(* Logix 5000 project; controller STAT 1756-L72 rev 20.12; software revision 20.04; part 34 of 34 *)
(* tags used below, declared in another part *)
   B3 : DINT[50];
   F8 : REAL[200];
   I1_000_Bit09 : ALIAS FOR stock:1:I.Point_9;
   I1_000_Bit10 : ALIAS FOR stock:1:I.Point_10;
   I2_000_Bit13 : ALIAS FOR stock:2:I.Point_13;   // chaudière colmatageLigne 30= on 1= off
   I2_000_Bit14 : ALIAS FOR stock:2:I.Point_14;   // DEFAUT CHAUDIEREiwts
   N20 : DINT[100];
   N7 : DINT[255];
   nitric_occupe : BOOL;
   O3_000_Bit06 : ALIAS FOR stock:3:O.Point_6;   // lampe BP sur ligne p
   O3_000_Bit07 : ALIAS FOR stock:3:O.Point_7;
   ons11 : BOOL;
   S_bp_dmd_naoh : BOOL;
   S_ok_pmp_nitrique : BOOL;
   S_run_pmp_nitrique : BOOL;
   T4 : TIMER[50];
   apport_soude_ibt_occupe : BOOL;
   dmd_soude_ibt_ok : BOOL;
   I19_001_Bit07 : ALIAS FOR I19[1].7;   // vanne soude de stock ouverte
   I19_001_Bit08 : ALIAS FOR I19[1].8;   // vanne soude de stock fermée
   L1_stat : DINT[20];
   L2_STAT : DINT[20];
   L3_STAT : DINT[20];
   lancystock1 : DINT;
   lancystock2 : DINT;
   MSG_R_L4 : MESSAGE;
   MSG_W_L4 : MESSAGE;
   mw2 : BOOL;
   N : INT[255];
   O16 : INT[2];
   onS14 : BOOL;
   onS15 : BOOL;
   onS16 : BOOL;
   S_def_airco_hT_l1 : BOOL;
   S_def_ventilo_hT_l1 : BOOL;
   S_naoh_ibt : BOOL;
   S_stock_v_naoh_f : BOOL;
   S_stock_v_naoh_o : BOOL;
   soude_ibt_fini : BOOL;
   stat_L1 : DINT[20];
   STAT_L2 : DINT[20];
   STAT_L3 : DINT[20];
   stocklancy1 : DINT;
   stocklancy2 : DINT;
   stocklancy4 : DINT;   // alarme lvl 1 stock
   stocklancy5 : DINT;   // alarme lvl 2 stock
   t1sec : TIMER;
(* stock, continued *)

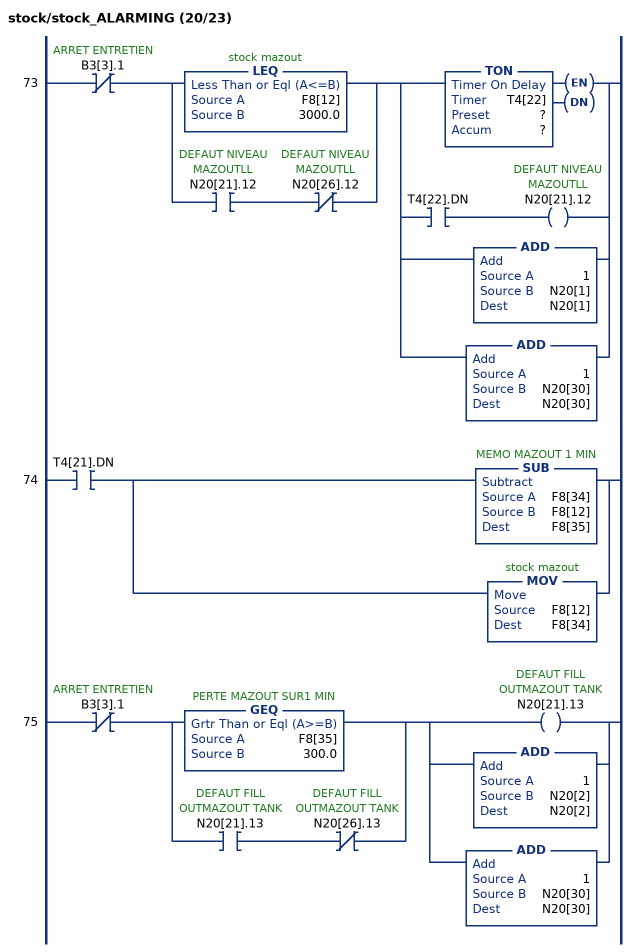
   [picture p698: stock/stock_ALARMING rungs 73-75]
   73: XIO(B3[3].1)[LEQ(F8[12],3000.0) ,XIC(N20[21].12) XIO(N20[26].12) ][TON(T4[22],?,?) ,XIC(T4[22].DN) OTE(N20[21].12) ,ADD(1,N20[1],N20[1]) ,ADD(1,N20[30],N20[30]) ];
   74: XIC(T4[21].DN)[SUB(F8[34],F8[12],F8[35]) ,MOV(F8[12],F8[34]) ];
   75: XIO(B3[3].1)[GEQ(F8[35],300.0) ,XIC(N20[21].13) XIO(N20[26].13) ][OTE(N20[21].13) ,ADD(1,N20[2],N20[2]) ,ADD(1,N20[30],N20[30]) ];
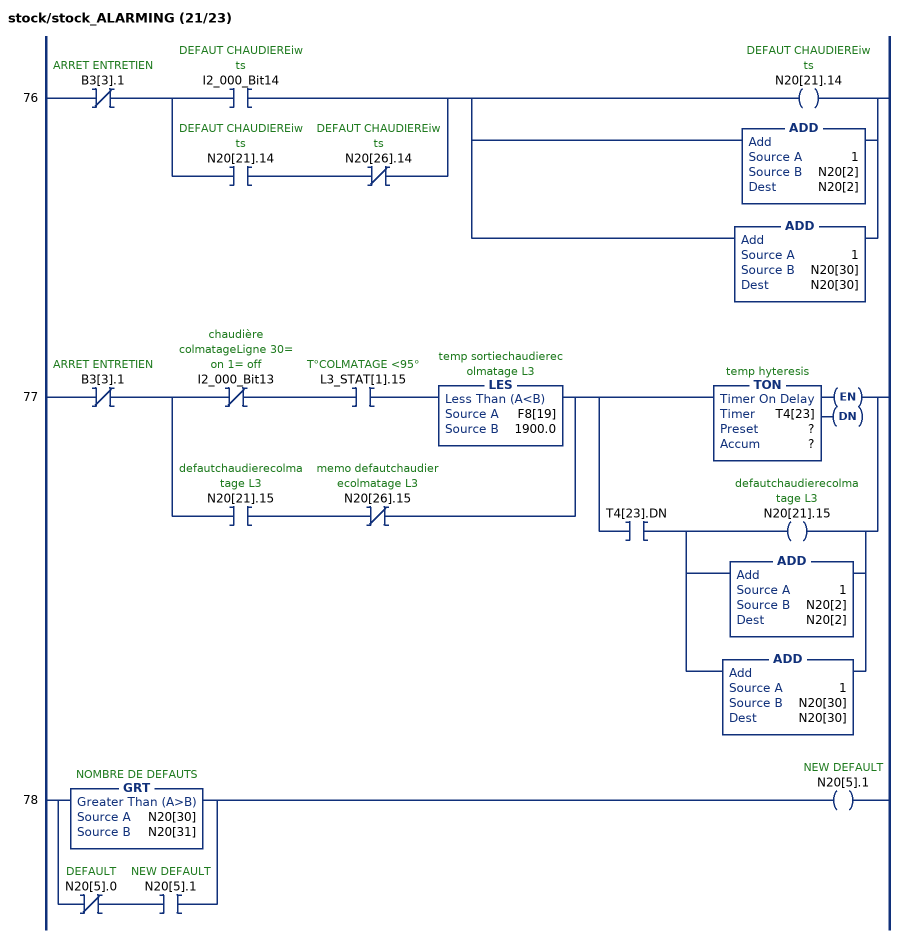
   76: XIO(B3[3].1)[XIC(I2_000_Bit14) ,XIC(N20[21].14) XIO(N20[26].14) ][OTE(N20[21].14) ,ADD(1,N20[2],N20[2]) ,ADD(1,N20[30],N20[30]) ];
   77: XIO(B3[3].1)[XIO(I2_000_Bit13) XIC(L3_STAT[1].15) LES(F8[19],1900.0) ,XIC(N20[21].15) XIO(N20[26].15) ][TON(T4[23],?,?) ,XIC(T4[23].DN) [OTE(N20[21].15) ,ADD(1,N20[2],N20[2]) ,ADD(1,N20[30],N20[30]) ] ];
   78: [GRT(N20[30],N20[31]) ,XIO(N20[5].0) XIC(N20[5].1) ]OTE(N20[5].1);
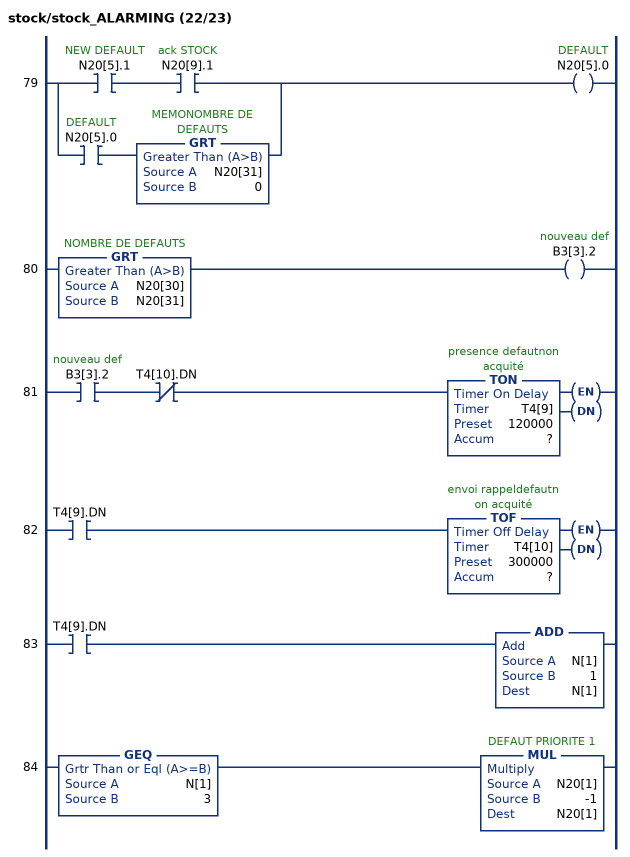
   79: [XIC(N20[5].1) XIC(N20[9].1) ,XIC(N20[5].0) GRT(N20[31],0) ]OTE(N20[5].0);
   80: GRT(N20[30],N20[31])OTE(B3[3].2);
   81: XIC(B3[3].2)XIO(T4[10].DN)TON(T4[9],?,?);
   82: XIC(T4[9].DN)TOF(T4[10],?,?);
   83: XIC(T4[9].DN)ADD(N[1],1,N[1]);
   84: GEQ(N[1],3)MUL(N20[1],-1,N20[1]);
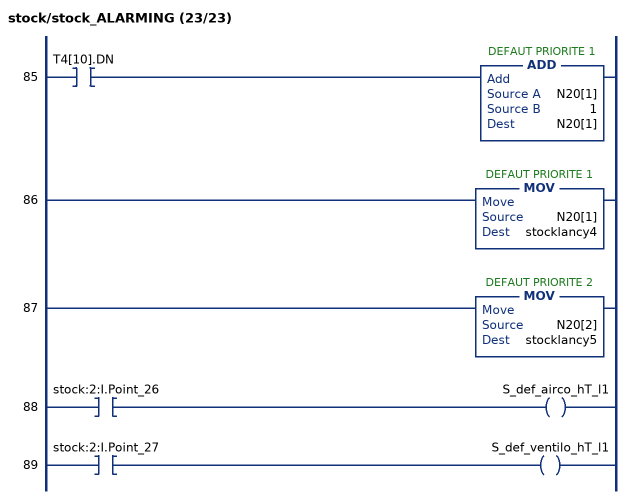
   85: XIC(T4[10].DN)ADD(N20[1],1,N20[1]);
   86: MOV(N20[1],stocklancy4);
   87: MOV(N20[2],stocklancy5);
   88: XIC(stock:2:I.Point_26)OTE(S_def_airco_hT_l1);
   89: XIC(stock:2:I.Point_27)OTE(S_def_ventilo_hT_l1);
END_ROUTINE

ROUTINE stock_nitric   (* ladder *)
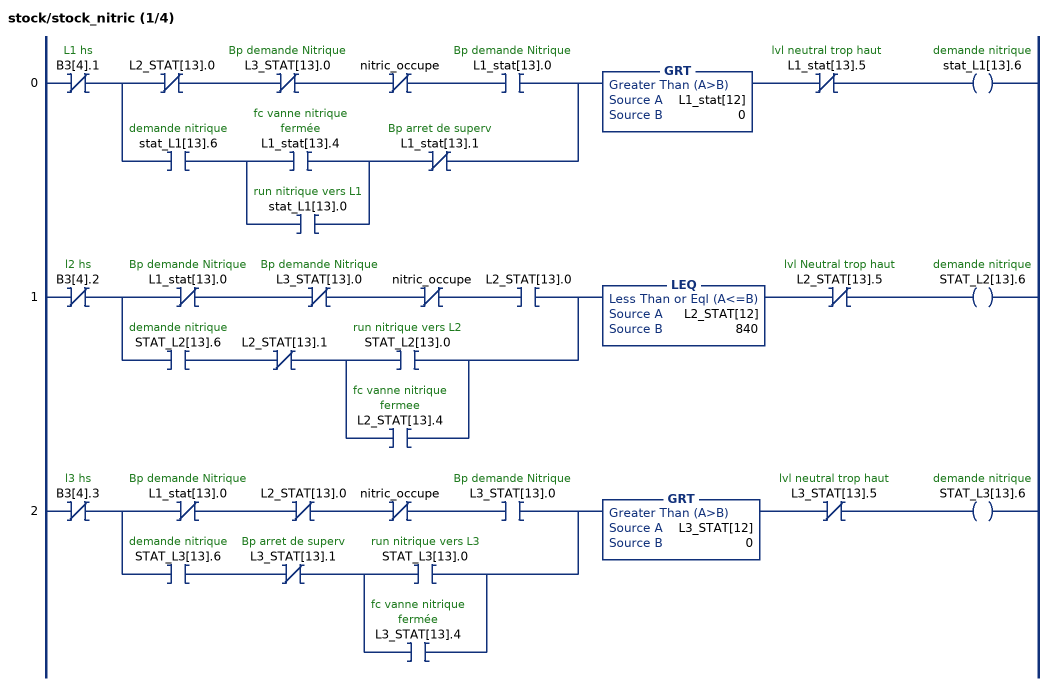
   0: XIO(B3[4].1)[XIO(L2_STAT[13].0) XIO(L3_STAT[13].0) XIO(nitric_occupe) XIC(L1_stat[13].0) ,XIC(stat_L1[13].6) [XIC(L1_stat[13].4) ,XIC(stat_L1[13].0) ] XIO(L1_stat[13].1) ]GRT(L1_stat[12],0)XIO(L1_stat[13].5)OTE(stat_L1[13].6);
   1: XIO(B3[4].2)[XIO(L1_stat[13].0) XIO(L3_STAT[13].0) XIO(nitric_occupe) XIC(L2_STAT[13].0) ,XIC(STAT_L2[13].6) XIO(L2_STAT[13].1) [XIC(STAT_L2[13].0) ,XIC(L2_STAT[13].4) ] ]LEQ(L2_STAT[12],840)XIO(L2_STAT[13].5)OTE(STAT_L2[13].6);
   2: XIO(B3[4].3)[XIO(L1_stat[13].0) XIO(L2_STAT[13].0) XIO(nitric_occupe) XIC(L3_STAT[13].0) ,XIC(STAT_L3[13].6) XIO(L3_STAT[13].1) [XIC(STAT_L3[13].0) ,XIC(L3_STAT[13].4) ] ]GRT(L3_STAT[12],0)XIO(L3_STAT[13].5)OTE(STAT_L3[13].6);
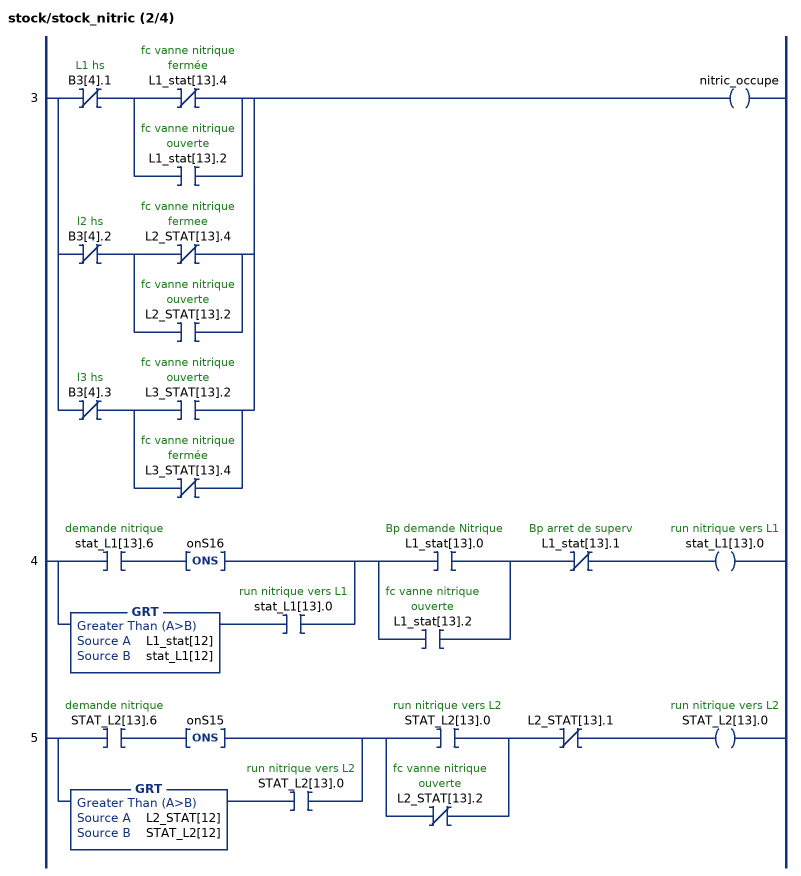
   3: [XIO(B3[4].1) [XIO(L1_stat[13].4) ,XIC(L1_stat[13].2) ] ,XIO(B3[4].2) [XIO(L2_STAT[13].4) ,XIC(L2_STAT[13].2) ] ,XIO(B3[4].3) [XIC(L3_STAT[13].2) ,XIO(L3_STAT[13].4) ] ]OTE(nitric_occupe);
   4: [XIC(stat_L1[13].6) ONS(onS16) ,GRT(L1_stat[12],stat_L1[12]) XIC(stat_L1[13].0) ][XIC(L1_stat[13].0) ,XIC(L1_stat[13].2) ]XIO(L1_stat[13].1)OTE(stat_L1[13].0);
   5: [XIC(STAT_L2[13].6) ONS(onS15) ,GRT(L2_STAT[12],STAT_L2[12]) XIC(STAT_L2[13].0) ][XIC(STAT_L2[13].0) ,XIO(L2_STAT[13].2) ]XIO(L2_STAT[13].1)OTE(STAT_L2[13].0);
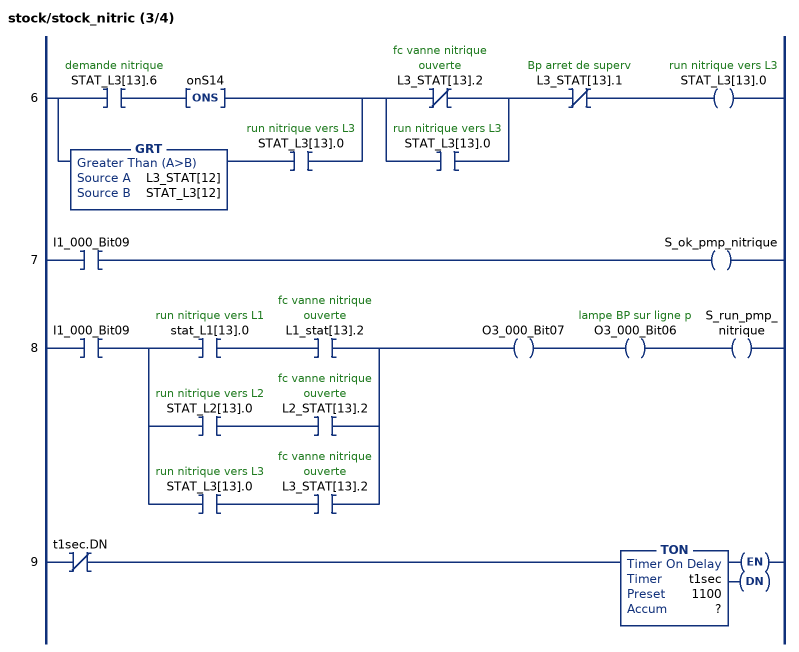
   6: [XIC(STAT_L3[13].6) ONS(onS14) ,GRT(L3_STAT[12],STAT_L3[12]) XIC(STAT_L3[13].0) ][XIO(L3_STAT[13].2) ,XIC(STAT_L3[13].0) ]XIO(L3_STAT[13].1)OTE(STAT_L3[13].0);
   7: XIC(I1_000_Bit09)OTE(S_ok_pmp_nitrique);
   8: XIC(I1_000_Bit09)[XIC(stat_L1[13].0) XIC(L1_stat[13].2) ,XIC(STAT_L2[13].0) XIC(L2_STAT[13].2) ,XIC(STAT_L3[13].0) XIC(L3_STAT[13].2) ]OTE(O3_000_Bit07)OTE(O3_000_Bit06)OTE(S_run_pmp_nitrique);
   9: XIO(t1sec.DN)TON(t1sec,?,?);
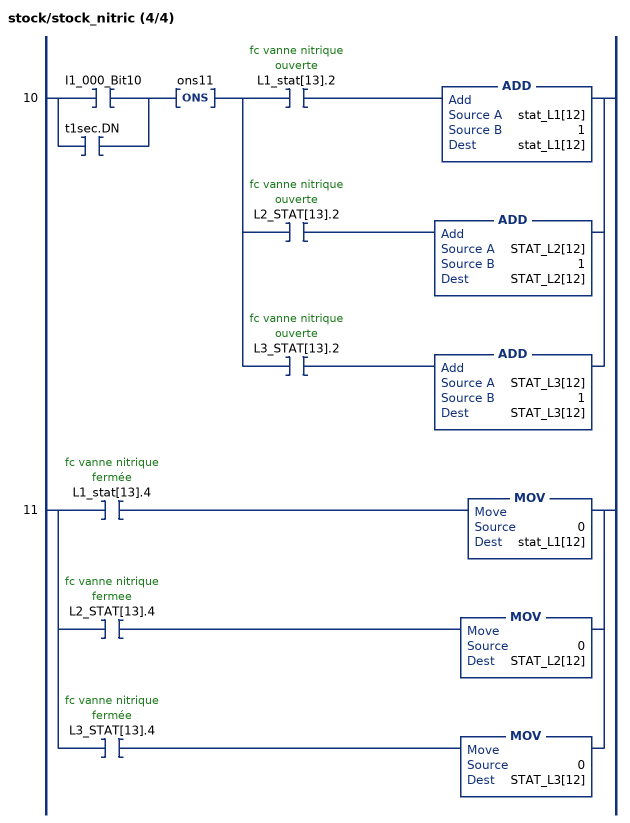
   10: [XIC(I1_000_Bit10) ,XIC(t1sec.DN) ]ONS(ons11)[XIC(L1_stat[13].2) ADD(stat_L1[12],1,stat_L1[12]) ,XIC(L2_STAT[13].2) ADD(STAT_L2[12],1,STAT_L2[12]) ,XIC(L3_STAT[13].2) ADD(STAT_L3[12],1,STAT_L3[12]) ];
   11: [XIC(L1_stat[13].4) MOV(0,stat_L1[12]) ,XIC(L2_STAT[13].4) MOV(0,STAT_L2[12]) ,XIC(L3_STAT[13].4) MOV(0,STAT_L3[12]) ];
END_ROUTINE

ROUTINE stock_SOUDE   (* ladder *)
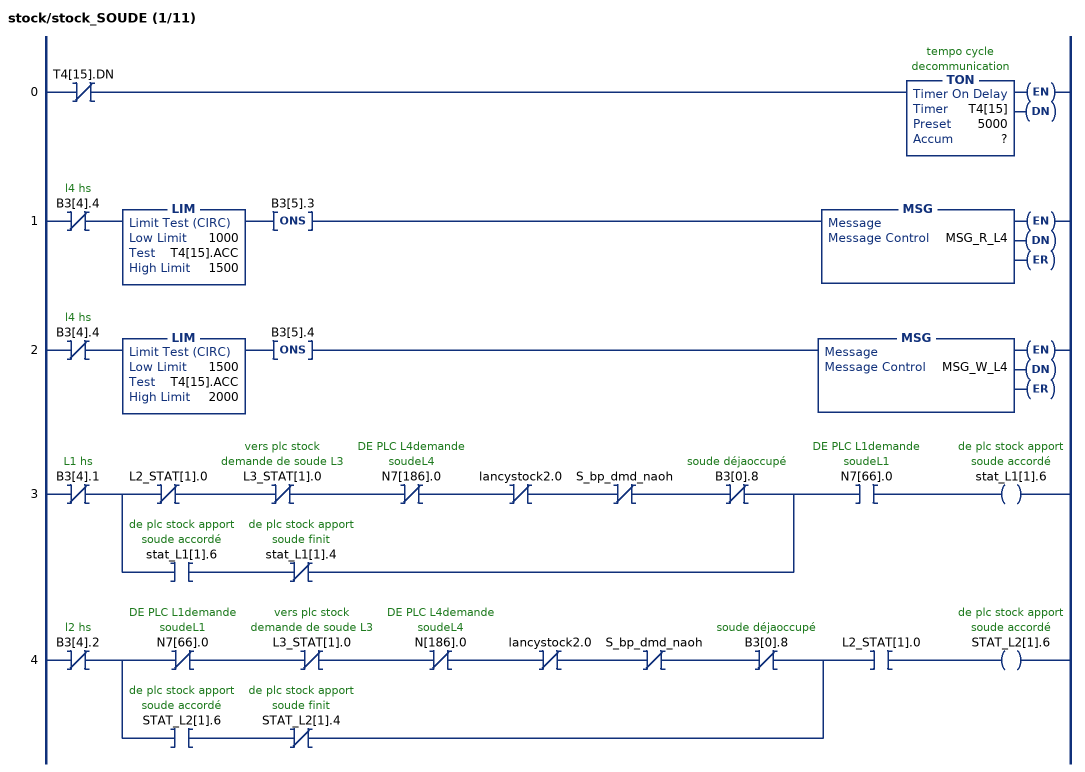
   0: XIO(T4[15].DN)TON(T4[15],?,?);
   1: XIO(B3[4].4)LIM(1000,T4[15].ACC,1500)ONS(B3[5].3)MSG(MSG_R_L4);
   2: XIO(B3[4].4)LIM(1500,T4[15].ACC,2000)ONS(B3[5].4)MSG(MSG_W_L4);
   3: XIO(B3[4].1)[XIO(L2_STAT[1].0) XIO(L3_STAT[1].0) XIO(N7[186].0) XIO(lancystock2.0) XIO(S_bp_dmd_naoh) XIO(B3[0].8) ,XIC(stat_L1[1].6) XIO(stat_L1[1].4) ]XIC(N7[66].0)OTE(stat_L1[1].6);
   4: XIO(B3[4].2)[XIO(N7[66].0) XIO(L3_STAT[1].0) XIO(N[186].0) XIO(lancystock2.0) XIO(S_bp_dmd_naoh) XIO(B3[0].8) ,XIC(STAT_L2[1].6) XIO(STAT_L2[1].4) ]XIC(L2_STAT[1].0)OTE(STAT_L2[1].6);
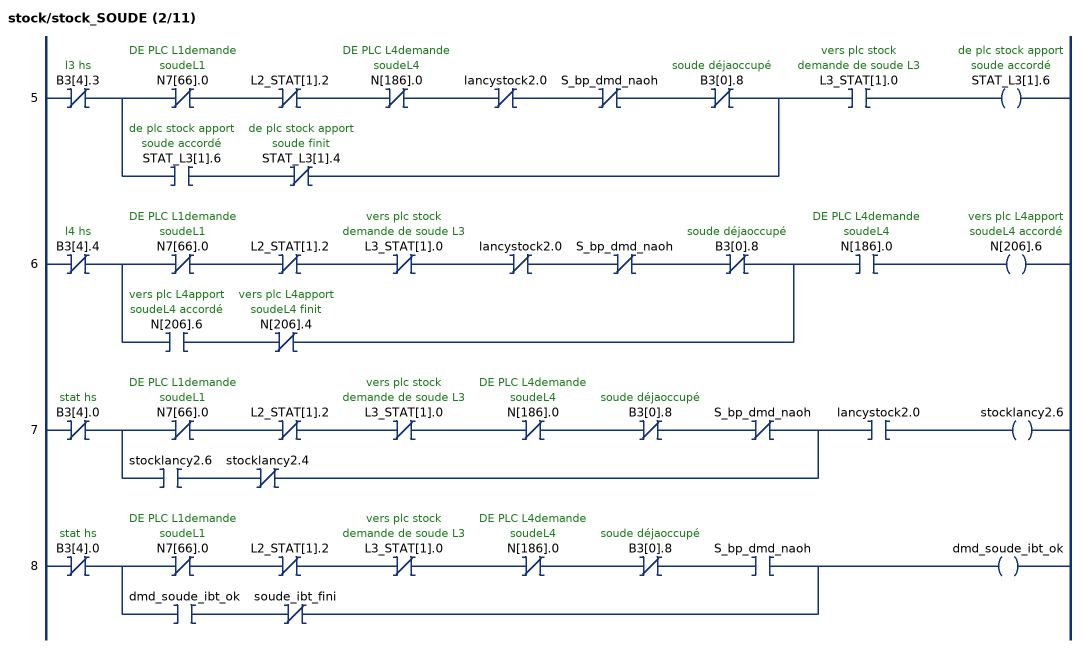
   5: XIO(B3[4].3)[XIO(N7[66].0) XIO(L2_STAT[1].2) XIO(N[186].0) XIO(lancystock2.0) XIO(S_bp_dmd_naoh) XIO(B3[0].8) ,XIC(STAT_L3[1].6) XIO(STAT_L3[1].4) ]XIC(L3_STAT[1].0)OTE(STAT_L3[1].6);
   6: XIO(B3[4].4)[XIO(N7[66].0) XIO(L2_STAT[1].2) XIO(L3_STAT[1].0) XIO(lancystock2.0) XIO(S_bp_dmd_naoh) XIO(B3[0].8) ,XIC(N[206].6) XIO(N[206].4) ]XIC(N[186].0)OTE(N[206].6);
   7: XIO(B3[4].0)[XIO(N7[66].0) XIO(L2_STAT[1].2) XIO(L3_STAT[1].0) XIO(N[186].0) XIO(B3[0].8) XIO(S_bp_dmd_naoh) ,XIC(stocklancy2.6) XIO(stocklancy2.4) ]XIC(lancystock2.0)OTE(stocklancy2.6);
   8: XIO(B3[4].0)[XIO(N7[66].0) XIO(L2_STAT[1].2) XIO(L3_STAT[1].0) XIO(N[186].0) XIO(B3[0].8) XIC(S_bp_dmd_naoh) ,XIC(dmd_soude_ibt_ok) XIO(soude_ibt_fini) ]OTE(dmd_soude_ibt_ok);
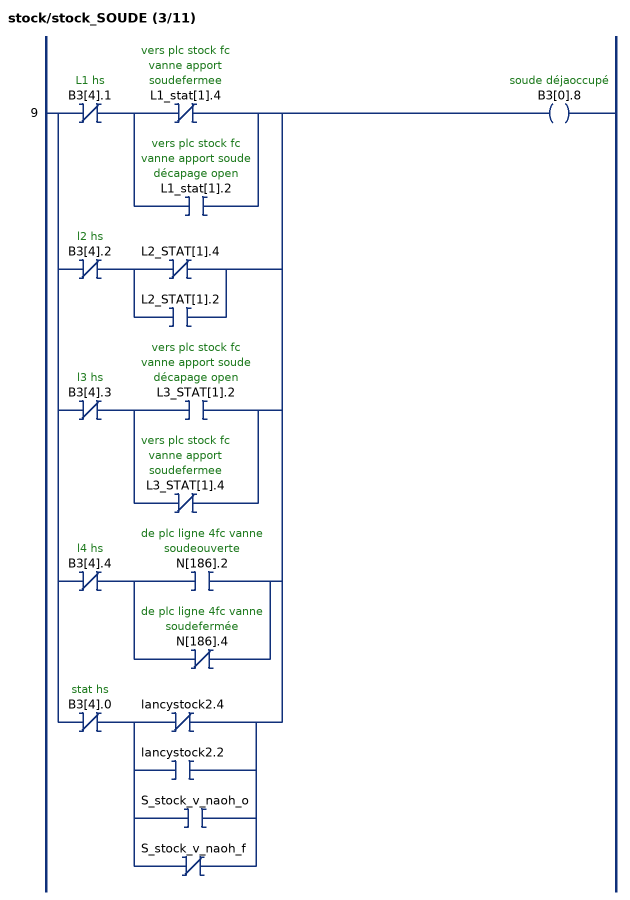
   9: [XIO(B3[4].1) [XIO(L1_stat[1].4) ,XIC(L1_stat[1].2) ] ,XIO(B3[4].2) [XIO(L2_STAT[1].4) ,XIC(L2_STAT[1].2) ] ,XIO(B3[4].3) [XIC(L3_STAT[1].2) ,XIO(L3_STAT[1].4) ] ,XIO(B3[4].4) [XIC(N[186].2) ,XIO(N[186].4) ] ,XIO(B3[4].0) [XIO(lancystock2.4) ,XIC(lancystock2.2) ,XIC(S_stock_v_naoh_o) ,XIO(S_stock_v_naoh_f) ] ]OTE(B3[0].8);
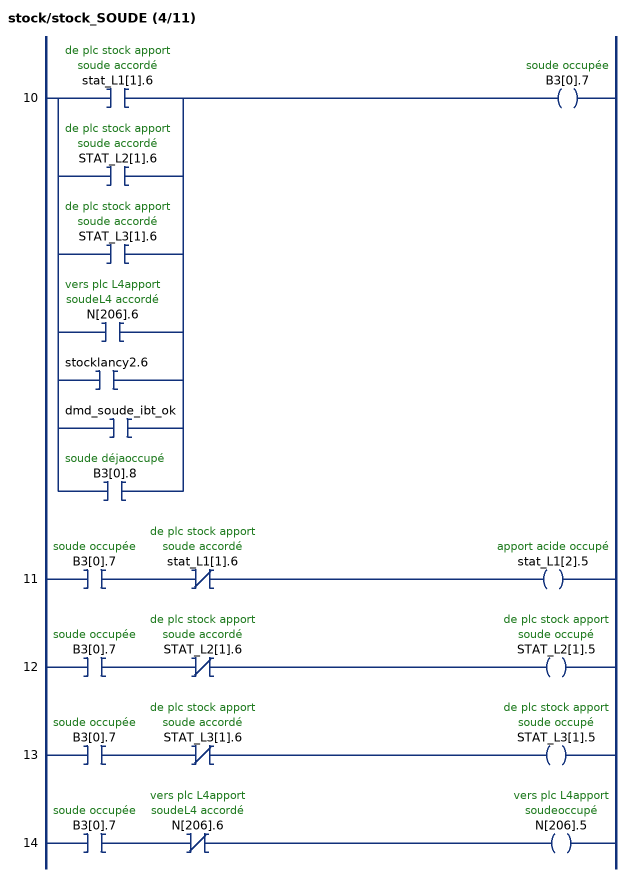
   10: [XIC(stat_L1[1].6) ,XIC(STAT_L2[1].6) ,XIC(STAT_L3[1].6) ,XIC(N[206].6) ,XIC(stocklancy2.6) ,XIC(dmd_soude_ibt_ok) ,XIC(B3[0].8) ]OTE(B3[0].7);
   11: XIC(B3[0].7)XIO(stat_L1[1].6)OTE(stat_L1[2].5);
   12: XIC(B3[0].7)XIO(STAT_L2[1].6)OTE(STAT_L2[1].5);
   13: XIC(B3[0].7)XIO(STAT_L3[1].6)OTE(STAT_L3[1].5);
   14: XIC(B3[0].7)XIO(N[206].6)OTE(N[206].5);
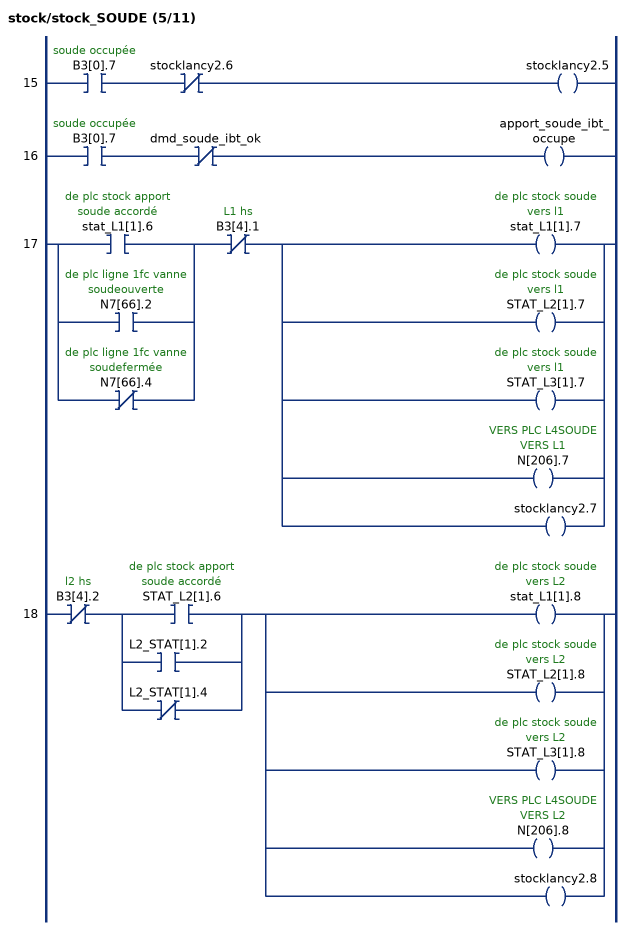
   15: XIC(B3[0].7)XIO(stocklancy2.6)OTE(stocklancy2.5);
   16: XIC(B3[0].7)XIO(dmd_soude_ibt_ok)OTE(apport_soude_ibt_occupe);
   17: [XIC(stat_L1[1].6) ,XIC(N7[66].2) ,XIO(N7[66].4) ]XIO(B3[4].1)[OTE(stat_L1[1].7) ,OTE(STAT_L2[1].7) ,OTE(STAT_L3[1].7) ,OTE(N[206].7) ,OTE(stocklancy2.7) ];
   18: XIO(B3[4].2)[XIC(STAT_L2[1].6) ,XIC(L2_STAT[1].2) ,XIO(L2_STAT[1].4) ][OTE(stat_L1[1].8) ,OTE(STAT_L2[1].8) ,OTE(STAT_L3[1].8) ,OTE(N[206].8) ,OTE(stocklancy2.8) ];
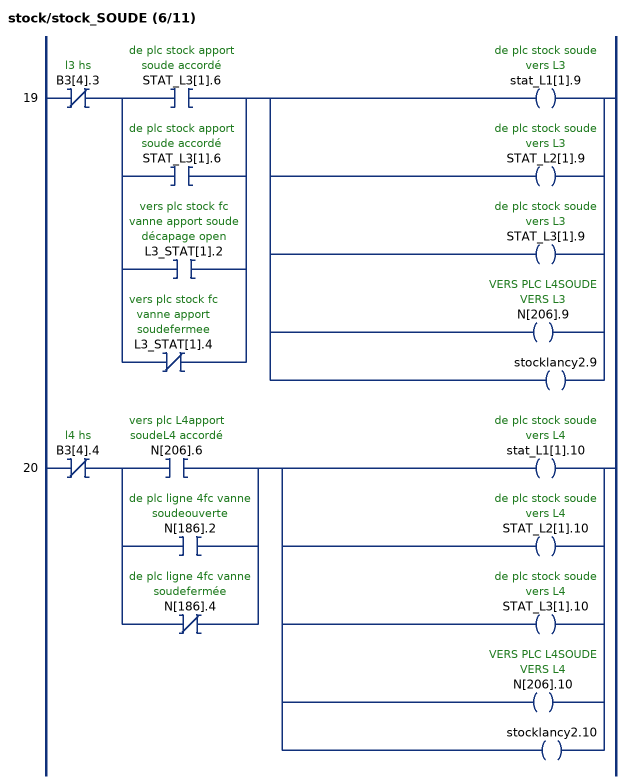
   19: XIO(B3[4].3)[XIC(STAT_L3[1].6) ,XIC(STAT_L3[1].6) ,XIC(L3_STAT[1].2) ,XIO(L3_STAT[1].4) ][OTE(stat_L1[1].9) ,OTE(STAT_L2[1].9) ,OTE(STAT_L3[1].9) ,OTE(N[206].9) ,OTE(stocklancy2.9) ];
   20: XIO(B3[4].4)[XIC(N[206].6) ,XIC(N[186].2) ,XIO(N[186].4) ][OTE(stat_L1[1].10) ,OTE(STAT_L2[1].10) ,OTE(STAT_L3[1].10) ,OTE(N[206].10) ,OTE(stocklancy2.10) ];
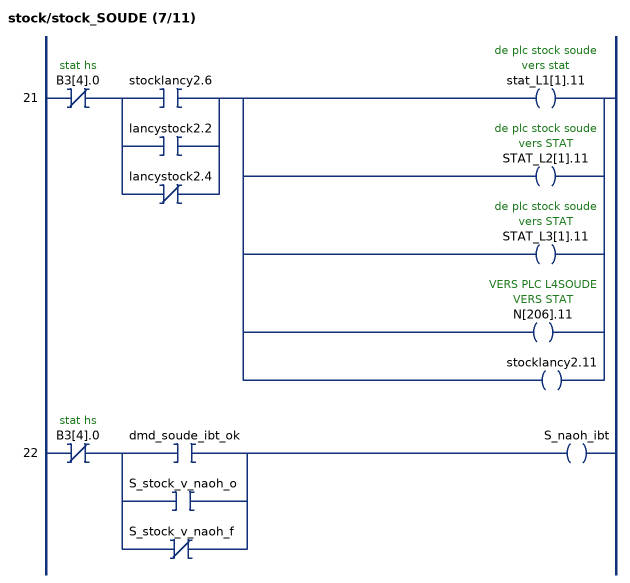
   21: XIO(B3[4].0)[XIC(stocklancy2.6) ,XIC(lancystock2.2) ,XIO(lancystock2.4) ][OTE(stat_L1[1].11) ,OTE(STAT_L2[1].11) ,OTE(STAT_L3[1].11) ,OTE(N[206].11) ,OTE(stocklancy2.11) ];
   22: XIO(B3[4].0)[XIC(dmd_soude_ibt_ok) ,XIC(S_stock_v_naoh_o) ,XIO(S_stock_v_naoh_f) ]OTE(S_naoh_ibt);
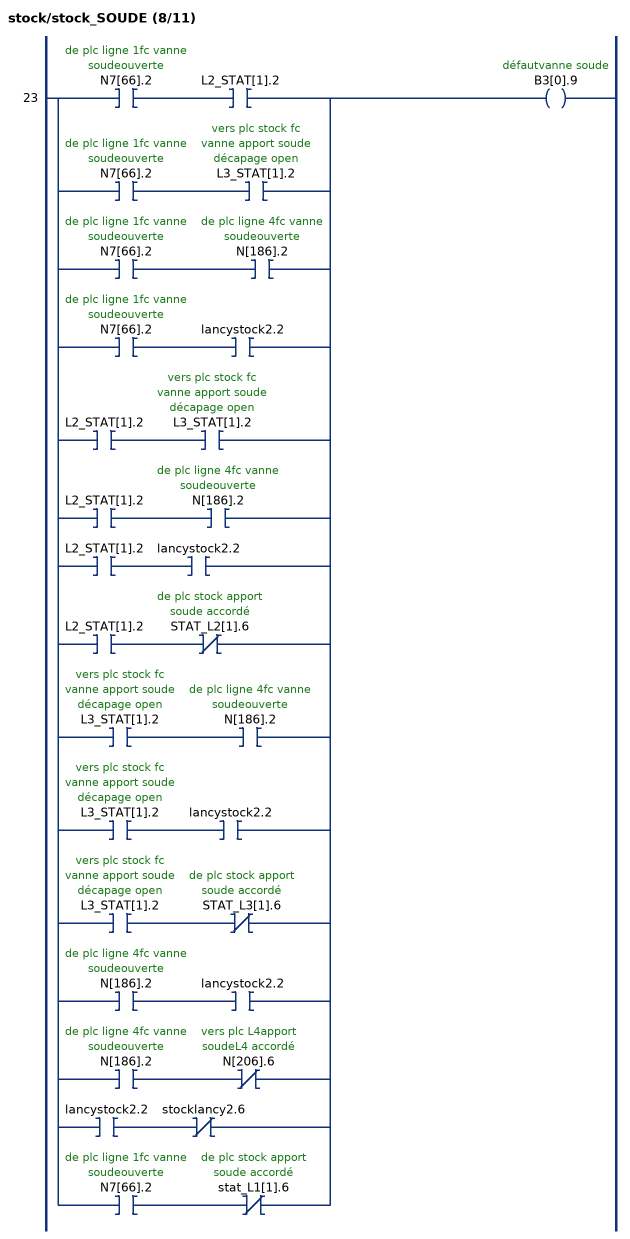
   23: [XIC(N7[66].2) XIC(L2_STAT[1].2) ,XIC(N7[66].2) XIC(L3_STAT[1].2) ,XIC(N7[66].2) XIC(N[186].2) ,XIC(N7[66].2) XIC(lancystock2.2) ,XIC(L2_STAT[1].2) XIC(L3_STAT[1].2) ,XIC(L2_STAT[1].2) XIC(N[186].2) ,XIC(L2_STAT[1].2) XIC(lancystock2.2) ,XIC(L2_STAT[1].2) XIO(STAT_L2[1].6) ,XIC(L3_STAT[1].2) XIC(N[186].2) ,XIC(L3_STAT[1].2) XIC(lancystock2.2) ,XIC(L3_STAT[1].2) XIO(STAT_L3[1].6) ,XIC(N[186].2) XIC(lancystock2.2) ,XIC(N[186].2) XIO(N[206].6) ,XIC(lancystock2.2) XIO(stocklancy2.6) ,XIC(N7[66].2) XIO(stat_L1[1].6) ]OTE(B3[0].9);
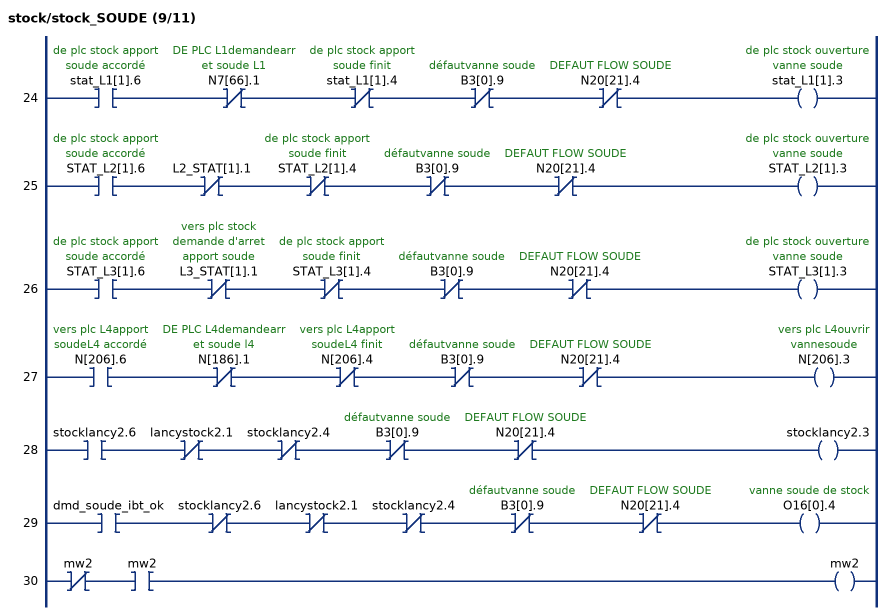
   24: XIC(stat_L1[1].6)XIO(N7[66].1)XIO(stat_L1[1].4)XIO(B3[0].9)XIO(N20[21].4)OTE(stat_L1[1].3);
   25: XIC(STAT_L2[1].6)XIO(L2_STAT[1].1)XIO(STAT_L2[1].4)XIO(B3[0].9)XIO(N20[21].4)OTE(STAT_L2[1].3);
   26: XIC(STAT_L3[1].6)XIO(L3_STAT[1].1)XIO(STAT_L3[1].4)XIO(B3[0].9)XIO(N20[21].4)OTE(STAT_L3[1].3);
   27: XIC(N[206].6)XIO(N[186].1)XIO(N[206].4)XIO(B3[0].9)XIO(N20[21].4)OTE(N[206].3);
   28: XIC(stocklancy2.6)XIO(lancystock2.1)XIO(stocklancy2.4)XIO(B3[0].9)XIO(N20[21].4)OTE(stocklancy2.3);
   29: XIC(dmd_soude_ibt_ok)XIO(stocklancy2.6)XIO(lancystock2.1)XIO(stocklancy2.4)XIO(B3[0].9)XIO(N20[21].4)OTE(O16[0].4);
   30: XIO(mw2)XIC(mw2)OTE(mw2);
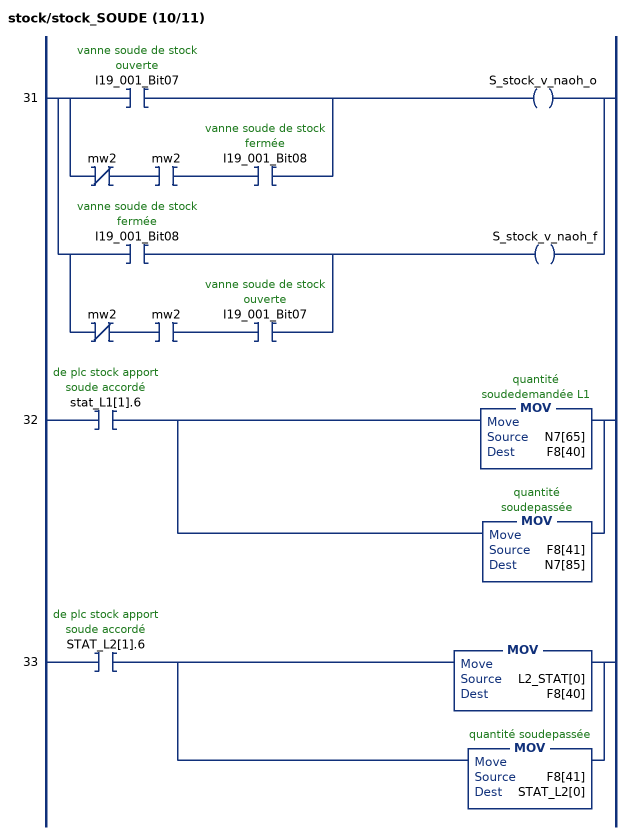
   31: [[XIC(I19_001_Bit07) ,XIO(mw2) XIC(mw2) XIC(I19_001_Bit08) ] OTE(S_stock_v_naoh_o) ,[XIC(I19_001_Bit08) ,XIO(mw2) XIC(mw2) XIC(I19_001_Bit07) ] OTE(S_stock_v_naoh_f) ];
   32: XIC(stat_L1[1].6)[MOV(N7[65],F8[40]) ,MOV(F8[41],N7[85]) ];
   33: XIC(STAT_L2[1].6)[MOV(L2_STAT[0],F8[40]) ,MOV(F8[41],STAT_L2[0]) ];
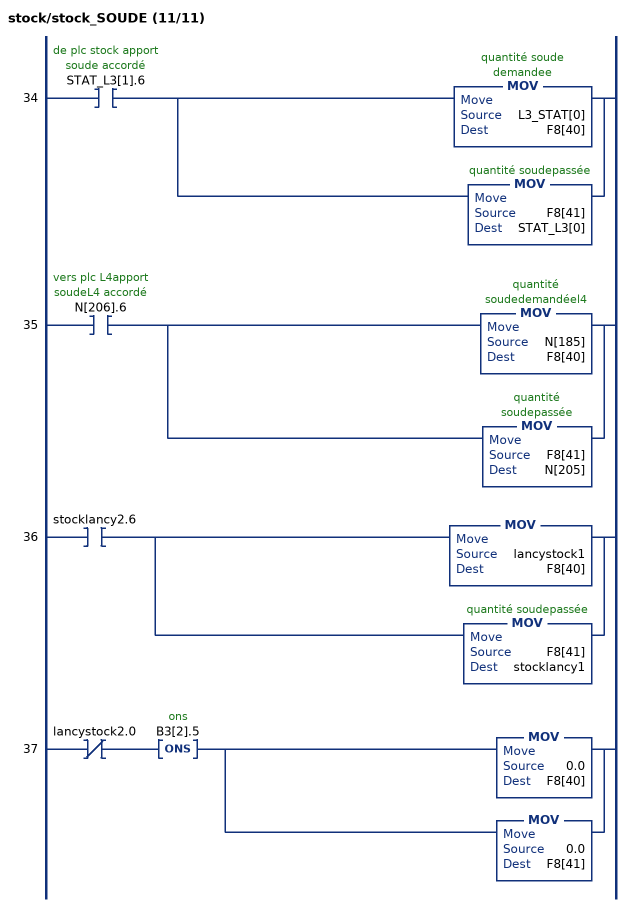
   34: XIC(STAT_L3[1].6)[MOV(L3_STAT[0],F8[40]) ,MOV(F8[41],STAT_L3[0]) ];
   35: XIC(N[206].6)[MOV(N[185],F8[40]) ,MOV(F8[41],N[205]) ];
   36: XIC(stocklancy2.6)[MOV(lancystock1,F8[40]) ,MOV(F8[41],stocklancy1) ];
   37: XIO(lancystock2.0)ONS(B3[2].5)[MOV(0.0,F8[40]) ,MOV(0.0,F8[41]) ];
END_ROUTINE
END_PROGRAM
